// TwinCAT 3 PLC project Untitled2
// ProgramVersion: 3.1.4024.0
// libraries:
//   Tc2_ModbusSrv, * (Beckhoff Automation GmbH)
//   Tc2_Standard, * (Beckhoff Automation GmbH)
//   Tc2_System, * (Beckhoff Automation GmbH)
//   Tc2_Utilities, * (Beckhoff Automation GmbH)
//   Tc3_Module, * (Beckhoff Automation GmbH)
// project tree:
//   GVLs/ Dataregs.TcGVL (not stored), Drum.TcGVL (not stored), IO.TcGVL (not stored), ModbusData.TcGVL (not stored), RobotDataIn.TcGVL (not stored), RobotDataOut.TcGVL (not stored), System.TcGVL
//   / PlcTask.TcTTO
//   POUs/ Drum_control.TcPOU (not stored), Fanuc_Start.TcPOU (not stored), FastTask.TcPOU (not stored), MAIN.TcPOU (not stored), Modbus_TCP.TcPOU (not stored), Robot.TcPOU (not stored)
// real-time tasks:
//   TASK PlcTask: cycle T#1ms, priority 20, ADS port 350
// I/O:
//   DEVICE Device 1 (Beckhoff CCAT)
//   DEVICE Device 2 (EtherCAT), AmsNetId 5.146.124.159.3.1
//     Term 7 (EK1200) [EK1200-5000 EtherCAT Power supply (2A E-Bus)]
//       Term 8 (EL1809) [EL1809 16Ch. Dig. Input 24V, 3ms]
//       Term 11 (EL2809) [EL2809 16Ch. Dig. Output 24V, 0.5A]
//       Term 1 (EL1918) [EL1918, 8Ch. Safety Input 24V, TwinSAFE]
//         modules: Module 2 (FSLOGIC)
//       Term 13 (EL2904) [EL2904, 4 Ch. Safety Output 24V, 0.5A, TwinSAFE]
//         modules: Module 1 (FSOES), Module 2 (DO)
//       Term 12 (EL9011) [EL9011 End Terminal]
//   DEVICE Device 3 (EtherCAT Automation Protocol), AmsNetId 5.146.124.159.4.1
//     Box 2 (Publisher)
//     Box 3 (Subscriber)
// variable links:
//   Device 2 (EtherCAT) <-> Device 2 (EtherCAT)/Term 7 (EK1200)/Term 1 (EL1918)
//     Term 7 (EK1200)/Term 13 (EL2904)/Module 1 (FSOES)/RxPDO/FSOE <-> ConnectionInputs/Message_31 TxPDO
//     Term 7 (EK1200)/Term 13 (EL2904)/Module 1 (FSOES)/TxPDO/FSOE <-> ConnectionOutputs/Message_31 RxPDO
//   Device 2 (EtherCAT) <-> Device 3 (EtherCAT Automation Protocol)/Box 2 (Publisher)
//     Term 7 (EK1200)/Term 1 (EL1918)/ConnectionInputs/Message_42 TxPDO <-> Pub-Var 1/Outputs/VarData
//   Device 2 (EtherCAT) <-> Device 3 (EtherCAT Automation Protocol)/Box 3 (Subscriber)
//     Term 7 (EK1200)/Term 1 (EL1918)/ConnectionOutputs/Message_42 RxPDO <-> Sub-Var 1/Inputs/VarData
//   Untitled2/Untitled2 Instance <-> Device 2 (EtherCAT)/Term 7 (EK1200)/Term 1 (EL1918)
//     PlcTask Inputs/IO.DI_AGV_EStop1 <-> Device Info Data/Internal I/O/Input Safe Data FSIN Module 2.Input
//     PlcTask Inputs/IO.DI_AGV_EStop2 <-> Device Info Data/Internal I/O/Input Safe Data FSIN Module 3.Input
//     PlcTask Inputs/IO.DI_Btn_ES <-> StandardInputs/Standard Out Var 38
//     PlcTask Inputs/IO.DI_Door_ES <-> StandardInputs/Standard Out Var 39
//     PlcTask Inputs/IO.DI_EStop <-> Device Info Data/Internal I/O/Input Safe Data FSIN Module 4.Input
//     PlcTask Inputs/IO.DI_SAFEoutput <-> Connection Info Data/Message_31 Info Data/Output Safe Data OutputChannel1
//     PlcTask Inputs/IO.DI_Touch1 <-> Device Info Data/Internal I/O/Input Safe Data FSIN Module 5.Input
//     PlcTask Inputs/IO.DI_Touch2 <-> Device Info Data/Internal I/O/Input Safe Data FSIN Module 6.Input
//     PlcTask Inputs/MAIN.COM_ERR <-> StandardInputs/Standard Out Var 40
//     PlcTask Inputs/MAIN.COM_ERR_S <-> StandardInputs/Standard Out Var 11
//     PlcTask Inputs/MAIN.FB_ERR <-> StandardInputs/Standard Out Var 43
//     PlcTask Inputs/MAIN.FB_ERR_S <-> StandardInputs/Standard Out Var 12
//     PlcTask Inputs/MAIN.OTHER_ERR <-> StandardInputs/Standard Out Var 41
//     PlcTask Inputs/MAIN.OTHER_ERR_S <-> StandardInputs/Standard Out Var 19
//     PlcTask Outputs/IO.DO_Btn_ES <-> StandardOutputs/Standard In Var 44
//     PlcTask Outputs/IO.DO_Door_ES <-> StandardOutputs/Standard In Var 45
//     PlcTask Outputs/IO.DO_RobotFault <-> StandardOutputs/Standard In Var 32
//     PlcTask Outputs/IO.DO_SafeEnble <-> StandardOutputs/Standard In Var 46
//     PlcTask Outputs/MAIN.ERR_ACK_S <-> StandardOutputs/Standard In Var 1
//     PlcTask Outputs/MAIN.RUN_S <-> StandardOutputs/Standard In Var 2
//     PlcTask Outputs/MAIN.Restart <-> StandardOutputs/Standard In Var 20
//   Untitled2/Untitled2 Instance <-> Device 2 (EtherCAT)/Term 7 (EK1200)/Term 11 (EL2809)
//     PlcTask Outputs/IO.DO_DrumallStop <-> Channel 5/Output
//     PlcTask Outputs/IO.DO_Light <-> Channel 6/Output
//     PlcTask Outputs/IO.DO_wheelBreak <-> Channel 10/Output
//   Untitled2/Untitled2 Instance <-> Device 2 (EtherCAT)/Term 7 (EK1200)/Term 8 (EL1809)
//     PlcTask Inputs/IO.DI_Drop{1..5} <-> Channel {7..11}/Input  (5 links)
//     PlcTask Inputs/IO.DI_Drum1 <-> Channel 4/Input
//     PlcTask Inputs/IO.DI_Reset_Button <-> Channel 13/Input
//     PlcTask Inputs/IO.DI_RobotFault <-> Channel 12/Input
//   Untitled2/Untitled2 Instance <-> Device 3 (EtherCAT Automation Protocol)/Box 2 (Publisher)
//     PlcTask Outputs/IO.DO_RUNStatus <-> Pub-Var 2/Outputs/VarData
//   Untitled2/Untitled2 Instance <-> Device 3 (EtherCAT Automation Protocol)/Box 3 (Subscriber)
//     PlcTask Inputs/IO.DI_Crawl <-> DoorDI/Inputs/VarData
//     PlcTask Inputs/IO.DI_DoorStatus <-> DoorStatus/Inputs/VarData
//     PlcTask Inputs/IO.DI_EStopStatus <-> EstopStatus/Inputs/VarData
//     PlcTask Inputs/IO.DI_SafeCrawl <-> EstopDI/Inputs/VarData

CONFIGURATION Untitled2
    RESOURCE PLC ON TwinCAT3
        TASK PlcTask(INTERVAL := T#1ms, PRIORITY := 20);
        PROGRAM MAIN WITH PlcTask : MAIN;
    END_RESOURCE
END_CONFIGURATION

// ---- GVLs/System.TcGVL
{attribute 'qualified_only'}
VAR_GLOBAL
	start :BOOL;
	stop :BOOL;
	reset :BOOL;
	pause :BOOL;
	restart :BOOL;
END_VAR
